{attribute 'qualified_only'}
// I/O Inputs from main application
//
VAR_GLOBAL

	// Input signals from main application...
	i_HtrON   AT %I*: BOOL; // Heater to ON
	i_Restart AT %I*: BOOL; // Restart simulation

END_VAR

(* stored: Version 1.1.0.1, ProductVersion 3.1.4022.6
   GVL IO_Inputs: Id {e3d782ef-84f8-4777-bb6d-4aa389da9db7} *)
